// TIA Portal V19 export
DATA_BLOCK "RO_2 DB"   // DB102
{ S7_Optimized_Access := 'FALSE' }
   VAR
      "RO-2 P-401A/B/C FEED PUMP" : Bool;
      "HPP-402 A" : Bool;
      "HPP-402 B" : Bool;
      "AGLV-401 RECIRC" : Bool;
      "AGLV-402 RECIRC" : Bool;
      "AGLV-401" : Bool;
      "AGLV-402" : Bool;
   END_VAR
BEGIN
END_DATA_BLOCK
